// TIA Portal project "TimesCont" (V14)
// Estudos de Times, Temporizadores e contadores

(* hardware
DEVICE "S7-1200 station_1"  S7-1200 Station
   slot 0: "Rack_0"  S7-1200 Rack  Rack  V1.0
   slot 1: "PLC_1_times"  CPU 1214C DC/DC/DC  6ES7 214-1AG40-0XB0  V4.2
*)

// ===== PLC "PLC_1_times"  CPU 1214C DC/DC/DC =====

VAR_GLOBAL   // PLC tag table "Default tag table"
   "System_Byte" AT %MB1 : Byte;
   "FirstScan" AT %M1.0 : Bool;
   "DiagStatusUpdate" AT %M1.1 : Bool;
   "AlwaysTRUE" AT %M1.2 : Bool;
   "AlwaysFALSE" AT %M1.3 : Bool;
   "Clock_Byte" AT %MB0 : Byte;
   "Clock_10Hz" AT %M0.0 : Bool;
   "Clock_5Hz" AT %M0.1 : Bool;
   "Clock_2.5Hz" AT %M0.2 : Bool;
   "Clock_2Hz" AT %M0.3 : Bool;
   "Clock_1.25Hz" AT %M0.4 : Bool;
   "Clock_1Hz" AT %M0.5 : Bool;
   "Clock_0.625Hz" AT %M0.6 : Bool;
   "Clock_0.5Hz" AT %M0.7 : Bool;
   "Tag_1" AT %M10.0 : Bool;
   "Tag_2" AT %M20.0 : Bool;
   "Tag_3" AT %M30.0 : Bool;
   "Tag_4" AT %M40.0 : Bool;
   "Tag_5" AT %M50.0 : Bool;
   "Tag_6" AT %M60.0 : Bool;
END_VAR

// folder: System blocks/Program resources

DATA_BLOCK "IEC_Timer_0_DB"   // DB1
{ S7_Optimized_Access := 'TRUE' }
AUTHOR : Simatic
FAMILY : IEC
NAME : IEC_TMR
VERSION : 1.0
// stored: InstanceOfName IEC_TIMER
"IEC_TIMER"
BEGIN
END_DATA_BLOCK

DATA_BLOCK "IEC_Timer_0_DB_1"   // DB2
{ S7_Optimized_Access := 'TRUE' }
AUTHOR : Simatic
FAMILY : IEC
NAME : IEC_TMR
VERSION : 1.0
// stored: InstanceOfName IEC_TIMER
"IEC_TIMER"
BEGIN
END_DATA_BLOCK

DATA_BLOCK "IEC_Timer_0_DB_2"   // DB3
{ S7_Optimized_Access := 'TRUE' }
AUTHOR : Simatic
FAMILY : IEC
NAME : IEC_TMR
VERSION : 1.0
// stored: InstanceOfName IEC_TIMER
"IEC_TIMER"
BEGIN
END_DATA_BLOCK

// folder: (top level)

FUNCTION "EstudoTimes" : Void   // FC1, LAD
TITLE = EstudoTimes TON
{ S7_Optimized_Access := 'TRUE' }
VERSION : 0.1
   VAR_TEMP
      CurrentTime : Time;
   END_VAR
BEGIN

REGION Network 1: TON
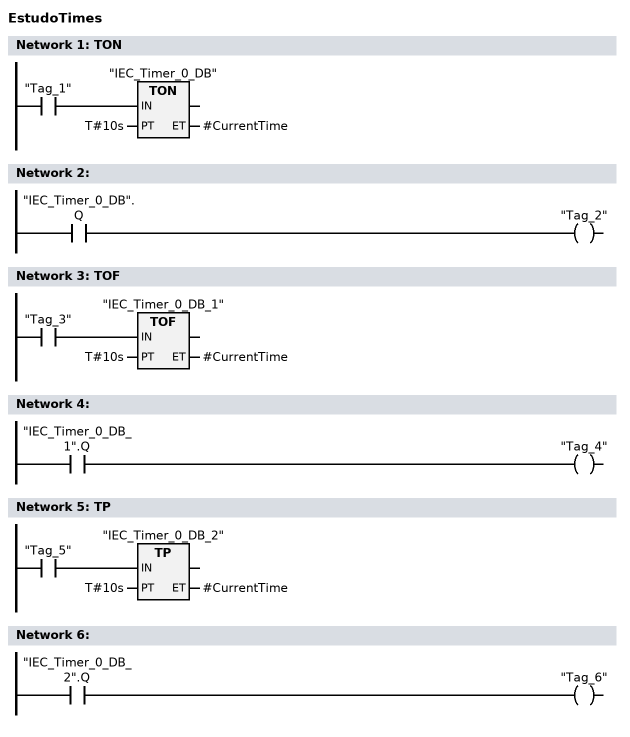
   "IEC_Timer_0_DB".TON(IN := "Tag_1", PT := T#10s, ET => #CurrentTime);
END_REGION

REGION Network 2
   RUNG wire#powerrail
      Contact( "IEC_Timer_0_DB".Q )
      Coil( "Tag_2" )
   END_RUNG
   // the same network as SCL:
   "Tag_2" := "IEC_Timer_0_DB".Q;
END_REGION

REGION Network 3: TOF
   "IEC_Timer_0_DB_1".TOF(IN := "Tag_3", PT := T#10s, ET => #CurrentTime);
END_REGION

REGION Network 4
   RUNG wire#powerrail
      Contact( "IEC_Timer_0_DB_1".Q )
      Coil( "Tag_4" )
   END_RUNG
   // the same network as SCL:
   "Tag_4" := "IEC_Timer_0_DB_1".Q;
END_REGION

REGION Network 5: TP
   "IEC_Timer_0_DB_2".TP(IN := "Tag_5", PT := T#10s, ET => #CurrentTime);
END_REGION

REGION Network 6
   RUNG wire#powerrail
      Contact( "IEC_Timer_0_DB_2".Q )
      Coil( "Tag_6" )
   END_RUNG
   // the same network as SCL:
   "Tag_6" := "IEC_Timer_0_DB_2".Q;
END_REGION
END_FUNCTION

ORGANIZATION_BLOCK "Main"   // OB1, LAD, ProgramCycle
TITLE = "Main Program Sweep (Cycle)"
{ S7_Optimized_Access := 'TRUE' }
VERSION : 0.1
   VAR_INPUT
      Initial_Call : Bool;   // Initial call of this OB
      Remanence : Bool;   // =True, if remanent data are available
   END_VAR
BEGIN

REGION Network 1
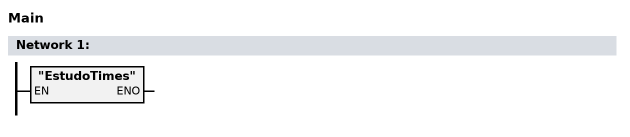
   RUNG wire#powerrail
      "EstudoTimes"()
   END_RUNG
   // the same network as SCL:
   "EstudoTimes"();
END_REGION
END_ORGANIZATION_BLOCK